# EPICS substitutions: modules/event/evrSupport/Db/ioc/IOC-IN20-AM01evr.substitutions
#==============================================================================
#
# Abs:  LCLS EVR IOC records for IN20 AM01
#
# Name: IOC-IN20-AM01evr.substitutions
#
#==============================================================================
#
file evrAMXX.db
{
pattern { DEVICE        }
	{ EVR:IN20:AM01 }
}
